(* PLC project Random_Generator, Unknown Unnamed 1 *)
(* stored: creationDateTime 2021-10-12T12:55:02, modificationDateTime 2022-08-16T15:46:52 *)

FUNCTION_BLOCK rand_generator
  VAR_INPUT
    IN : BOOL;
  END_VAR
  VAR
    M : BOOL := 0;
    INIT : BOOL := 0;
  END_VAR
  VAR_OUTPUT
    OUT : UDINT := 0;
  END_VAR

            (* This example uses Pragmas to write C code directly on *)
(* your Structured Text code *)

(* Some platforms require including <time.h> library *)
(* for this to work. If you get compilation errors, *)
(* just uncomment the declaration below *)
{//#include <time.h>}


(* Initialize our random generator *)
(* This IF is called only the first time this *)
(* block executes *)
IF INIT = 0 THEN
  {time_t t;
  srand((unsigned) time(&t))}
  INIT := 1;
END_IF;

IF M = 0 and IN = 1 THEN
  (* Using pragma to write code directly in C. *)
  (* You can access your PLC program variables using *)
  (* GetFbVar(var,...) and SetFbVar(var,val,...) calls *)
  {SetFbVar(OUT,rand())}
END_IF;
M := IN;
          
END_FUNCTION_BLOCK

PROGRAM Random
  VAR
    button : BOOL;
    value : UDINT;
    rand_generator0 : rand_generator;
  END_VAR

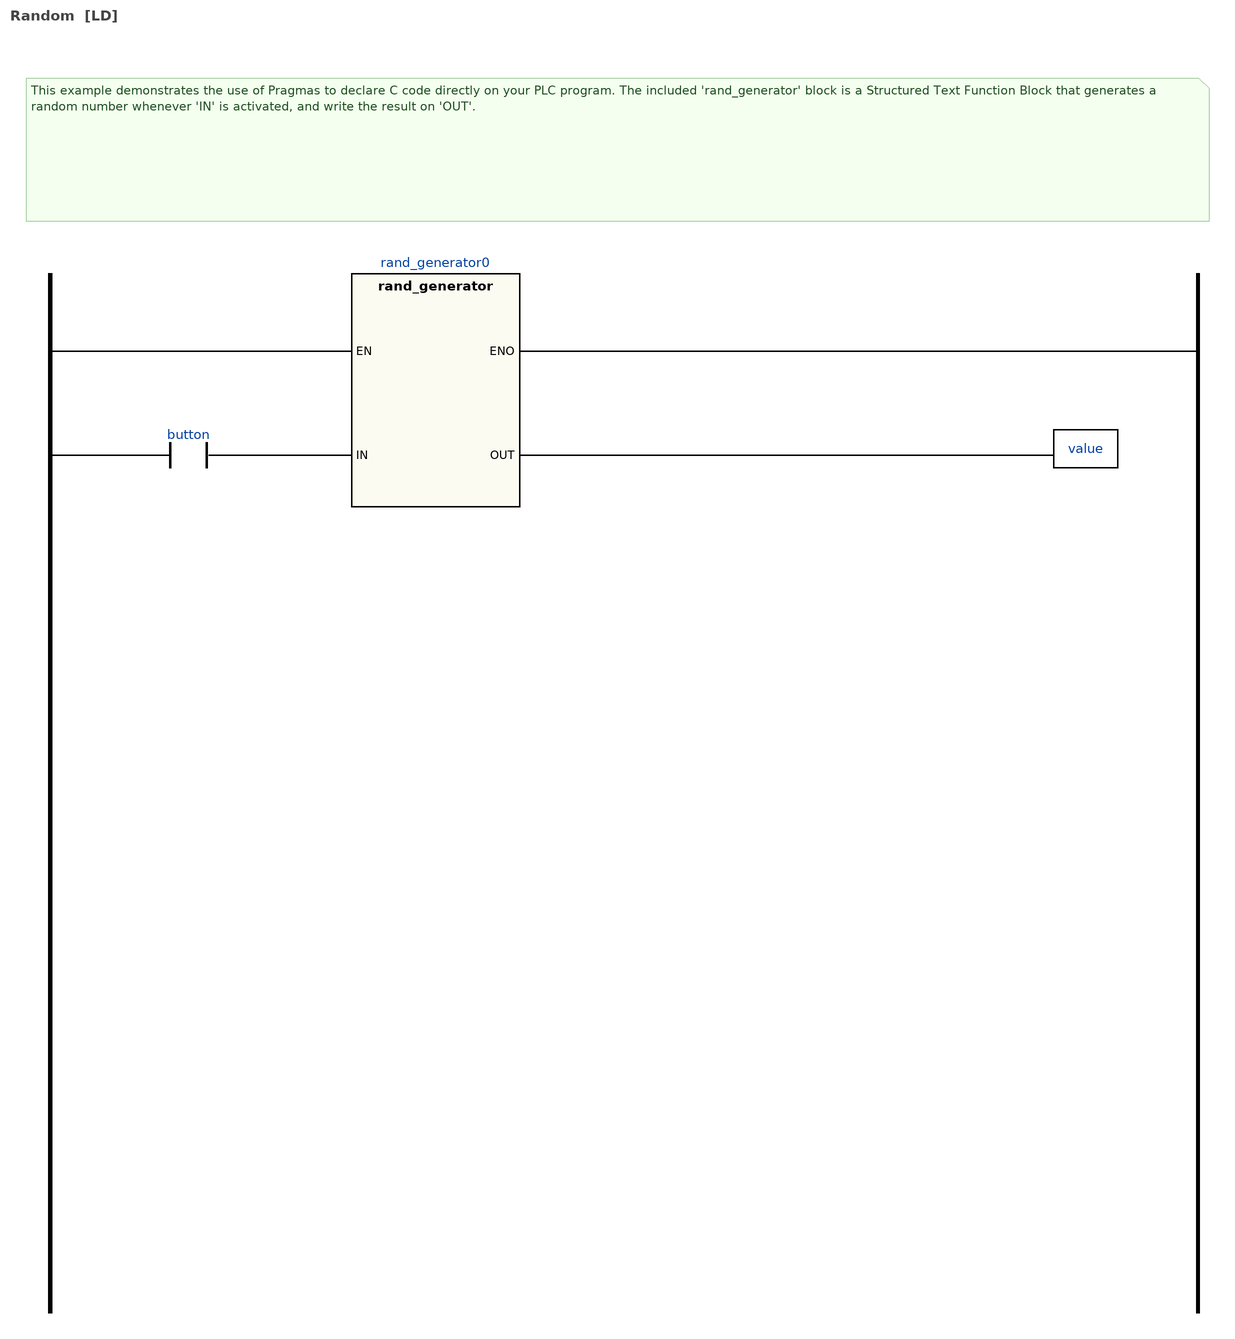
(* LD diagram, written out as Structured Text *)
(* This example demonstrates the use of Pragmas to declare C code directly on your PLC program. The included 'rand_generator' block is a Structured Text Function Block that generates a random number whenever 'IN' is activated, and write the result on 'OUT'. *)
rand_generator0(IN := button);
value := rand_generator0.OUT;
END_PROGRAM

CONFIGURATION Config0
  RESOURCE Res0 ON PLC
    TASK task0(INTERVAL := T#20ms, PRIORITY := 0);
    PROGRAM instance0 WITH task0 : Random;
  END_RESOURCE
END_CONFIGURATION
